% RSLogix 500 project alarm_count.RSS, saved by version 8.30.00.16 %
PROJECT "UNTITLED"    % processor: Bul.1763 MicroLogix 1100 Series B %

PROGRAM FILES
  LAD 2 "MAIN"  4 rungs
  LAD 3 "SUB_AND"  6 rungs
  LAD 4 "PARALLEL"  12 rungs
  LAD 5 "XIC_BRUTEF"  3 rungs
  LAD 6 "LOOKUPBYTE"  5 rungs
  LAD 7 "SUBANDUNRL"  129 rungs
  LAD 254 "WRITE_BITS"  5 rungs
  LAD 255 "BITSPRBYTE"  5 rungs

DATA FILES
  O0 OUTPUT  4 elements
  I1 INPUT  6 elements
  S2 STATUS  66 elements
  B3 BINARY  3 elements
  T4 TIMER  11 elements
  C5 COUNTER  1 elements
  R6 CONTROL  1 elements
  N7 INTEGER  10 elements
  F8 FLOAT  4 elements
  L9 LONG_DATA  12 elements
  N10 BITSPRBYTE  256 elements
  L11 LONG_MASKS  12 elements
  L100 CONTRLTIME  256 elements
  L101 SUBANDTIME  256 elements
  L102 PARLLLTIME  256 elements
  L103 XIC_TIME  256 elements
  L104 LOOKUPTIME  256 elements
  L105 SUBANDUNRL  256 elements

LADDER 2 "MAIN"
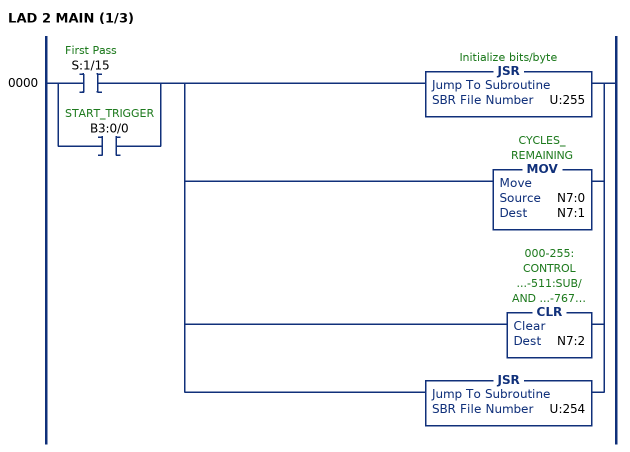
% Rung: 0 %
SOR BST XIC S:1/15 NXB XIC B3:0/0 BND BST JSR U:255 NXB MOV N7:0 N7:1 NXB CLR N7:2 NXB JSR U:254 BND EOR
%   S:1/15  "First Pass" %
%   B3:0/0  START_TRIGGER %
%   U:255  "Initialize bits/byte" %
%   N7:0  TEST_CYCLES %
%   N7:1  CYCLES_REMAINING %
%   N7:2  WHICH  "000-255:CONTROL ...-511:SUB/AND ...-767:PARALLEL ...-1023:XIC ...-1279:LOOKUP_BYTE" %

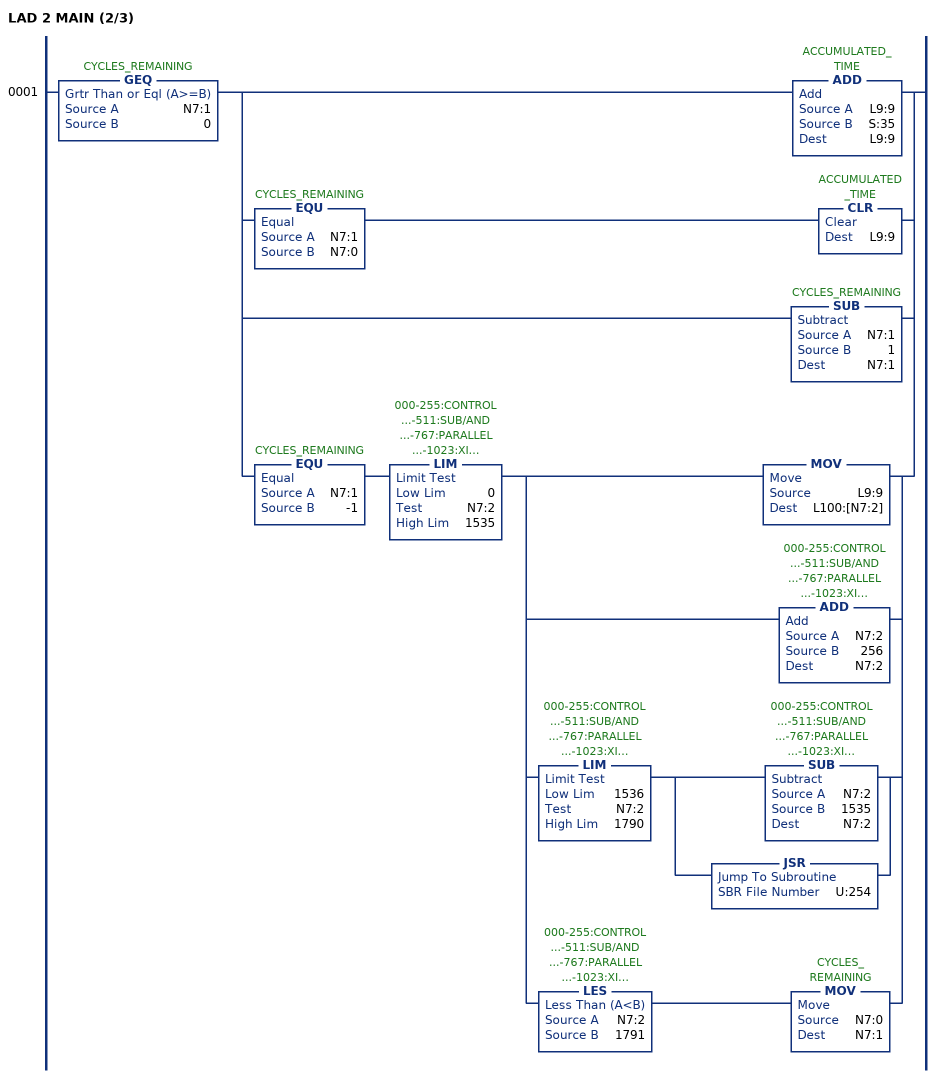
% Rung: 1 %
SOR GEQ N7:1 0 BST ADD L9:9 S:35 L9:9 NXB EQU N7:1 N7:0 CLR L9:9 NXB SUB N7:1 1 N7:1 NXB EQU N7:1 -1 LIM 0 N7:2 1535 BST MOV L9:9 L100:[N7:2] NXB ADD N7:2 256 N7:2 NXB LIM 1536 N7:2 1790 BST SUB N7:2 1535 N7:2 NXB JSR U:254 BND NXB LES N7:2 1791 MOV N7:0 N7:1 BND BND EOR
%   N7:1  CYCLES_REMAINING %
%   L9:9  ACCUMULATED_TIME %
%   S:35  "Last 1 ms Scan Time" %
%   N7:0  TEST_CYCLES %
%   N7:2  WHICH  "000-255:CONTROL ...-511:SUB/AND ...-767:PARALLEL ...-1023:XIC ...-1279:LOOKUP_BYTE" %

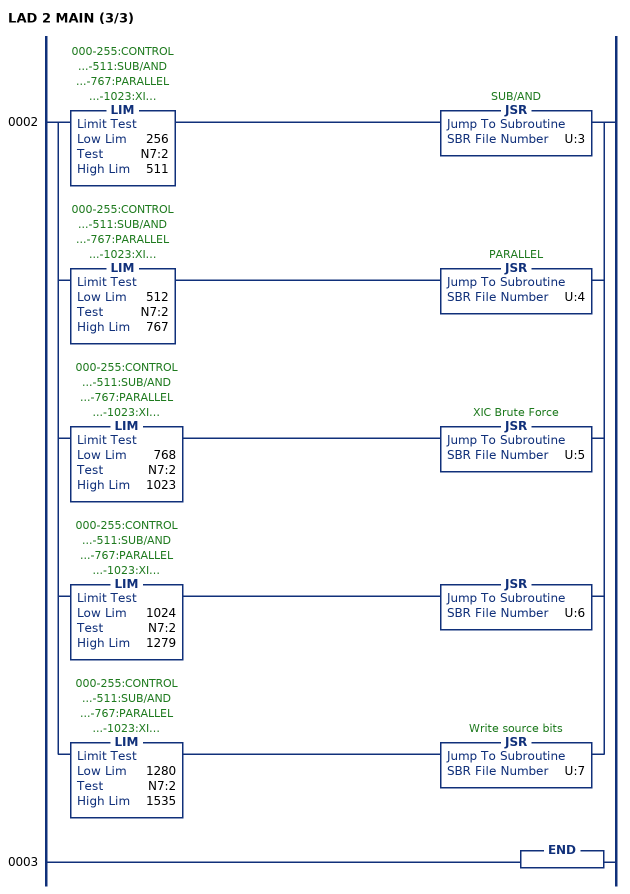
% Rung: 2 %
SOR BST LIM 256 N7:2 511 JSR U:3 NXB LIM 512 N7:2 767 JSR U:4 NXB LIM 768 N7:2 1023 JSR U:5 NXB LIM 1024 N7:2 1279 JSR U:6 NXB LIM 1280 N7:2 1535 JSR U:7 BND EOR
%   N7:2  WHICH  "000-255:CONTROL ...-511:SUB/AND ...-767:PARALLEL ...-1023:XIC ...-1279:LOOKUP_BYTE" %
%   U:3  "SUB/AND" %
%   U:4  "PARALLEL" %
%   U:5  "XIC Brute Force" %
%   U:7  "Write source bits" %
% Rung: 3 %
SOR END EOR

LADDER 3 "SUB_AND"
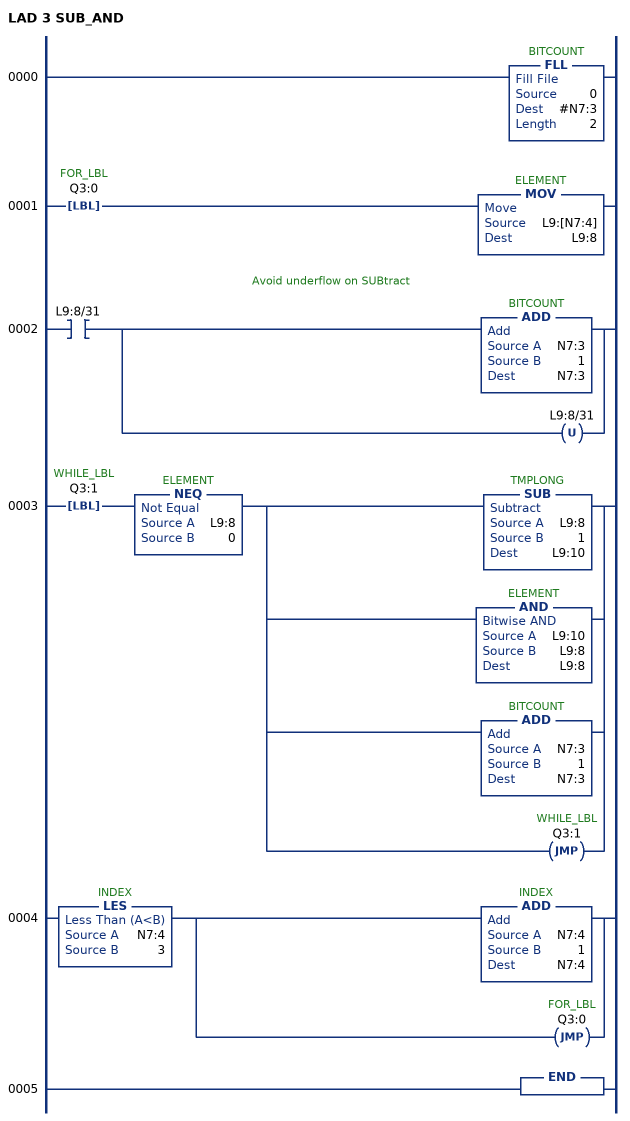
% Rung: 0 %
SOR FLL 0 #N7:3 2 EOR
%   N7:3  BITCOUNT %
% Rung: 1 %
SOR LBL Q3:0 MOV L9:[N7:4] L9:8 EOR
%   Q3:0  FOR_LBL %
%   N7:4  INDEX %
%   L9:8  ELEMENT %
% Rung: 2 %
% Avoid underflow on SUBtract %
SOR XIC L9:8/31 BST ADD N7:3 1 N7:3 NXB OTU L9:8/31 BND EOR
%   N7:3  BITCOUNT %
% Rung: 3 %
SOR LBL Q3:1 NEQ L9:8 0 BST SUB L9:8 1 L9:10 NXB AND L9:10 L9:8 L9:8 NXB ADD N7:3 1 N7:3 NXB JMP Q3:1 BND EOR
%   Q3:1  WHILE_LBL %
%   L9:8  ELEMENT %
%   L9:10  TMPLONG %
%   N7:3  BITCOUNT %
% Rung: 4 %
SOR LES N7:4 3 BST ADD N7:4 1 N7:4 NXB JMP Q3:0 BND EOR
%   N7:4  INDEX %
%   Q3:0  FOR_LBL %
% Rung: 5 %
SOR END EOR

LADDER 4 "PARALLEL"
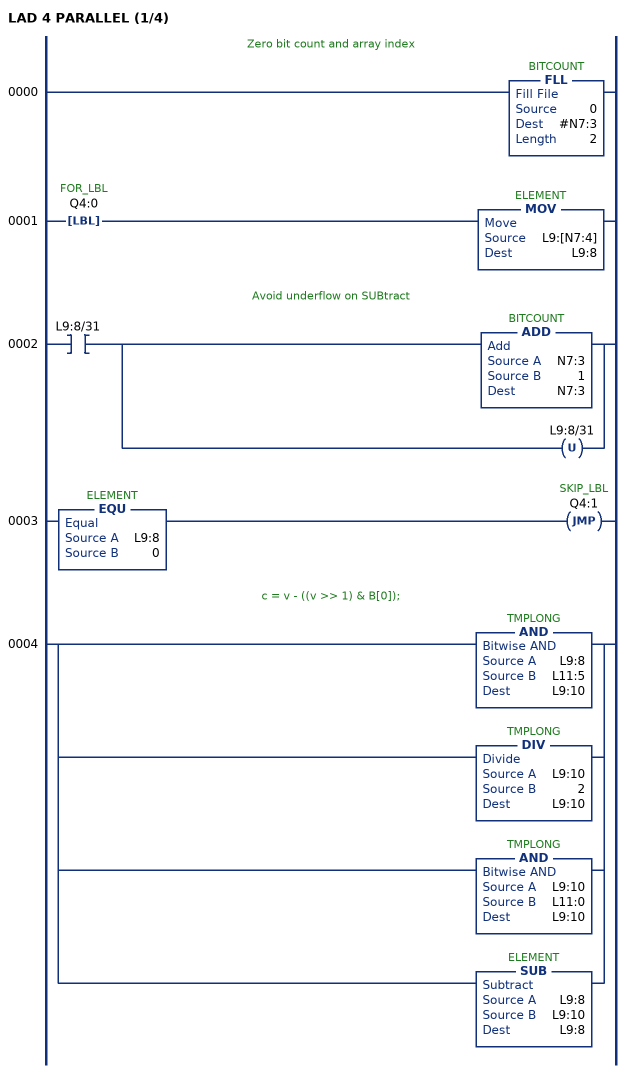
% Rung: 0 %
% Zero bit count and array index %
SOR FLL 0 #N7:3 2 EOR
%   N7:3  BITCOUNT %
% Rung: 1 %
SOR LBL Q4:0 MOV L9:[N7:4] L9:8 EOR
%   Q4:0  "FOR_LBL" %
%   N7:4  INDEX %
%   L9:8  ELEMENT %
% Rung: 2 %
% Avoid underflow on SUBtract %
SOR XIC L9:8/31 BST ADD N7:3 1 N7:3 NXB OTU L9:8/31 BND EOR
%   N7:3  BITCOUNT %
% Rung: 3 %
SOR EQU L9:8 0 JMP Q4:1 EOR
%   L9:8  ELEMENT %
%   Q4:1  "SKIP_LBL" %
% Rung: 4 %
% c = v - ((v >> 1) & B[0]); %
SOR BST AND L9:8 L11:5 L9:10 NXB DIV L9:10 2 L9:10 NXB AND L9:10 L11:0 L9:10 NXB SUB L9:8 L9:10 L9:8 BND EOR
%   L9:8  ELEMENT %
%   L11:5  0XFFFFFFFE_S0 %
%   L9:10  TMPLONG %
%   L11:0  0X55555555_B0 %

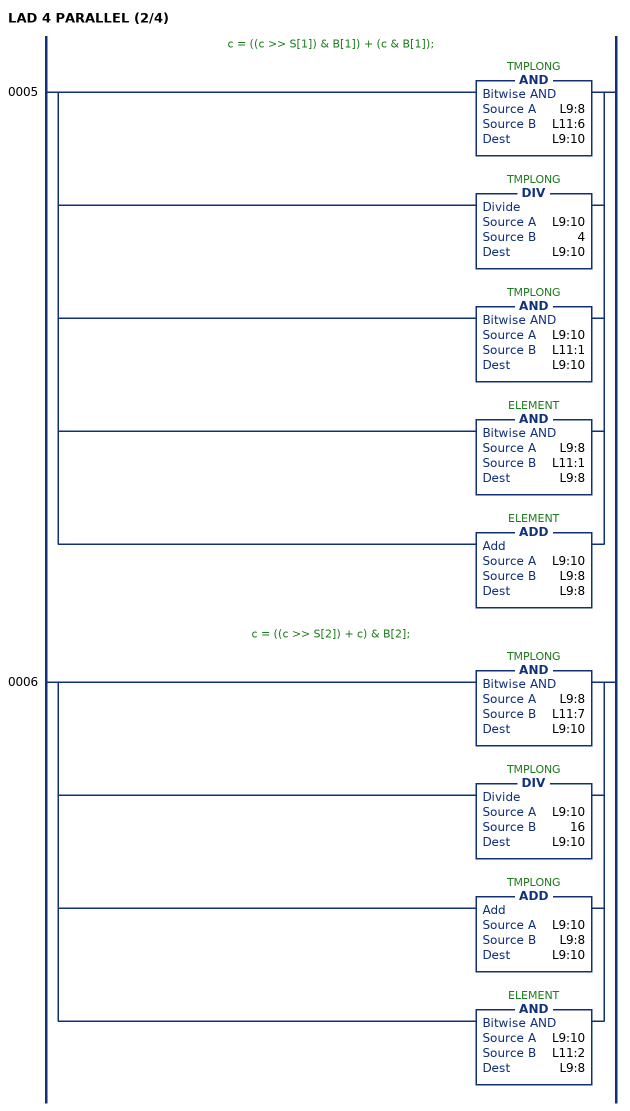
% Rung: 5 %
% c = ((c >> S[1]) & B[1]) + (c & B[1]); %
SOR BST AND L9:8 L11:6 L9:10 NXB DIV L9:10 4 L9:10 NXB AND L9:10 L11:1 L9:10 NXB AND L9:8 L11:1 L9:8 NXB ADD L9:10 L9:8 L9:8 BND EOR
%   L9:8  ELEMENT %
%   L11:6  0XFFFFFFFC_S1 %
%   L9:10  TMPLONG %
%   L11:1  0X33333333_B1 %
% Rung: 6 %
% c = ((c >> S[2]) + c) & B[2]; %
SOR BST AND L9:8 L11:7 L9:10 NXB DIV L9:10 16 L9:10 NXB ADD L9:10 L9:8 L9:10 NXB AND L9:10 L11:2 L9:8 BND EOR
%   L9:8  ELEMENT %
%   L11:7  0XFFFFFFF0_S2 %
%   L9:10  TMPLONG %
%   L11:2  0X0F0F0F0F_B2 %

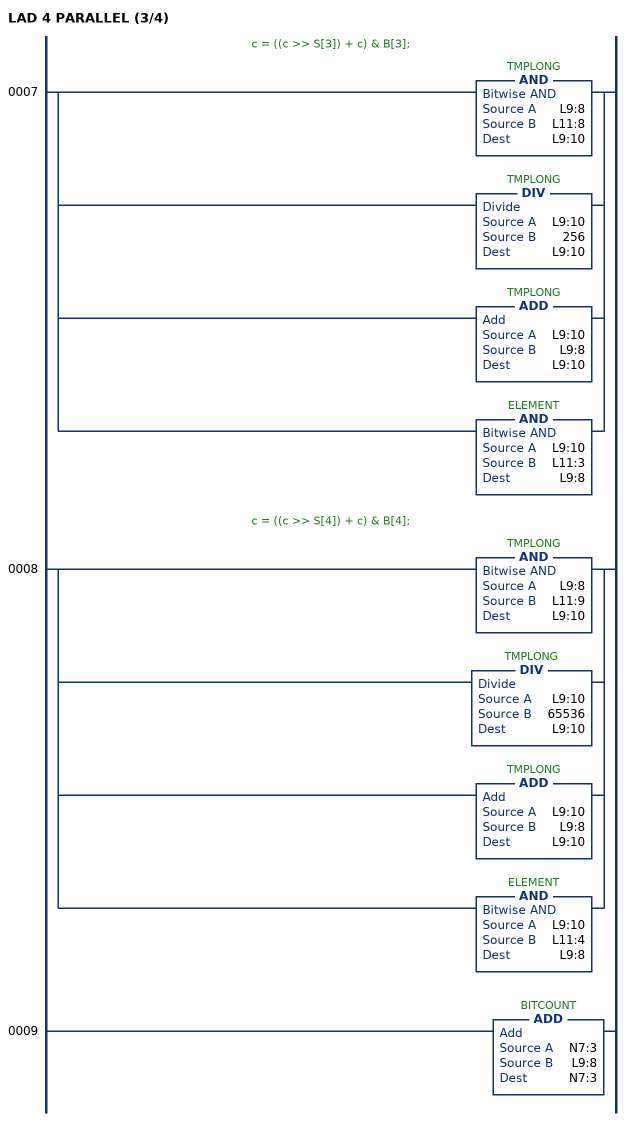
% Rung: 7 %
% c = ((c >> S[3]) + c) & B[3]; %
SOR BST AND L9:8 L11:8 L9:10 NXB DIV L9:10 256 L9:10 NXB ADD L9:10 L9:8 L9:10 NXB AND L9:10 L11:3 L9:8 BND EOR
%   L9:8  ELEMENT %
%   L11:8  0XFFFFFF00_S3 %
%   L9:10  TMPLONG %
%   L11:3  0X00FF00FF_B3 %
% Rung: 8 %
% c = ((c >> S[4]) + c) & B[4]; %
SOR BST AND L9:8 L11:9 L9:10 NXB DIV L9:10 65536 L9:10 NXB ADD L9:10 L9:8 L9:10 NXB AND L9:10 L11:4 L9:8 BND EOR
%   L9:8  ELEMENT %
%   L11:9  0XFFFF0000_S4 %
%   L9:10  TMPLONG %
%   L11:4  0X0000FFFF_B4 %
% Rung: 9 %
SOR ADD N7:3 L9:8 N7:3 EOR
%   N7:3  BITCOUNT %
%   L9:8  ELEMENT %

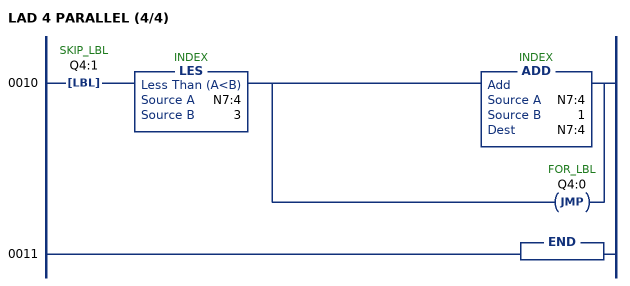
% Rung: 10 %
SOR LBL Q4:1 LES N7:4 3 BST ADD N7:4 1 N7:4 NXB JMP Q4:0 BND EOR
%   Q4:1  "SKIP_LBL" %
%   N7:4  INDEX %
%   Q4:0  "FOR_LBL" %
% Rung: 11 %
SOR END EOR

LADDER 5 "XIC_BRUTEF"
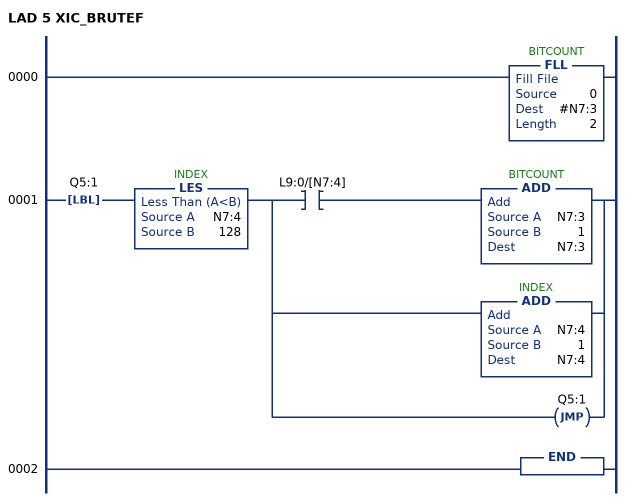
% Rung: 0 %
SOR FLL 0 #N7:3 2 EOR
%   N7:3  BITCOUNT %
% Rung: 1 %
SOR LBL Q5:1 LES N7:4 128 BST XIC L9:0/[N7:4] ADD N7:3 1 N7:3 NXB ADD N7:4 1 N7:4 NXB JMP Q5:1 BND EOR
%   N7:4  INDEX %
%   L9:0  128_SOURCE_BITS %
%   N7:3  BITCOUNT %
% Rung: 2 %
SOR END EOR

LADDER 6 "LOOKUPBYTE"
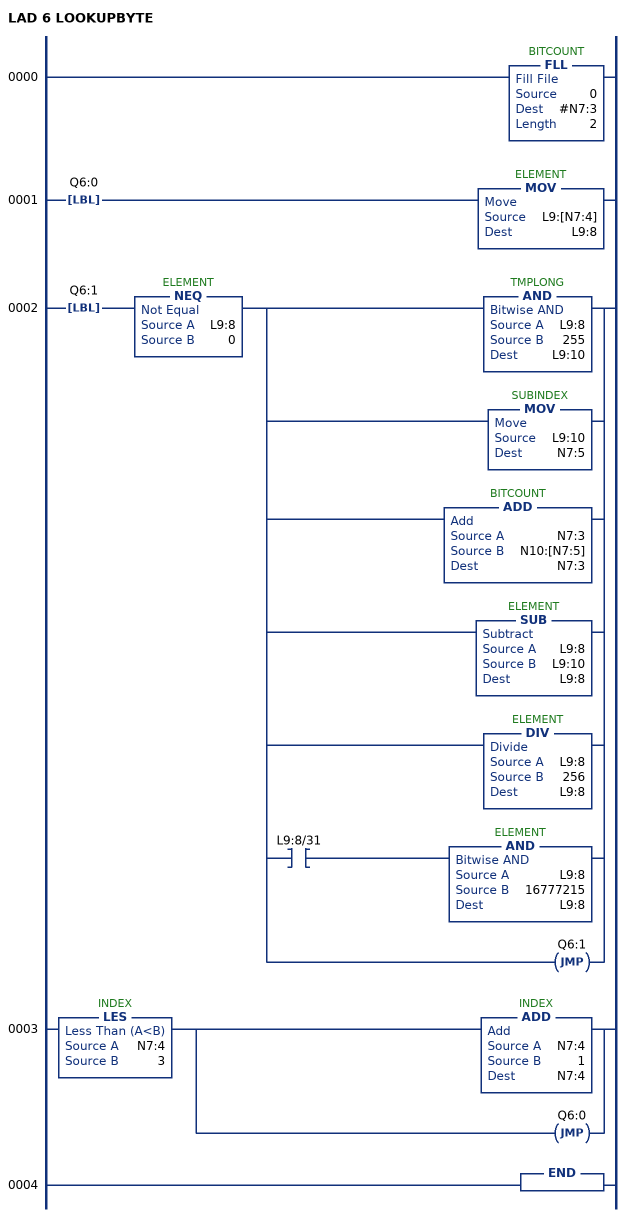
% Rung: 0 %
SOR FLL 0 #N7:3 2 EOR
%   N7:3  BITCOUNT %
% Rung: 1 %
SOR LBL Q6:0 MOV L9:[N7:4] L9:8 EOR
%   N7:4  INDEX %
%   L9:8  ELEMENT %
% Rung: 2 %
SOR LBL Q6:1 NEQ L9:8 0 BST AND L9:8 255 L9:10 NXB MOV L9:10 N7:5 NXB ADD N7:3 N10:[N7:5] N7:3 NXB SUB L9:8 L9:10 L9:8 NXB DIV L9:8 256 L9:8 NXB XIC L9:8/31 AND L9:8 16777215 L9:8 NXB JMP Q6:1 BND EOR
%   L9:8  ELEMENT %
%   L9:10  TMPLONG %
%   N7:5  SUBINDEX %
%   N7:3  BITCOUNT %
% Rung: 3 %
SOR LES N7:4 3 BST ADD N7:4 1 N7:4 NXB JMP Q6:0 BND EOR
%   N7:4  INDEX %
% Rung: 4 %
SOR END EOR

LADDER 7 "SUBANDUNRL"
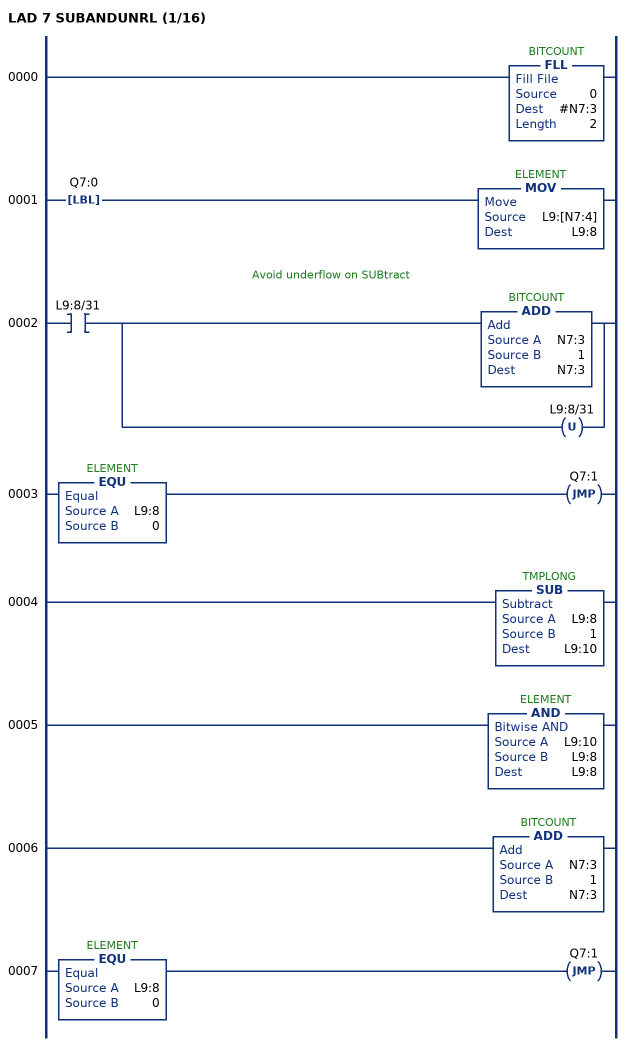
% Rung: 0 %
SOR FLL 0 #N7:3 2 EOR
%   N7:3  BITCOUNT %
% Rung: 1 %
SOR LBL Q7:0 MOV L9:[N7:4] L9:8 EOR
%   N7:4  INDEX %
%   L9:8  ELEMENT %
% Rung: 2 %
% Avoid underflow on SUBtract %
SOR XIC L9:8/31 BST ADD N7:3 1 N7:3 NXB OTU L9:8/31 BND EOR
%   N7:3  BITCOUNT %
% Rung: 3 %
SOR EQU L9:8 0 JMP Q7:1 EOR
%   L9:8  ELEMENT %
% Rung: 4 %
SOR SUB L9:8 1 L9:10 EOR
%   L9:8  ELEMENT %
%   L9:10  TMPLONG %
% Rung: 5 %
SOR AND L9:10 L9:8 L9:8 EOR
%   L9:10  TMPLONG %
%   L9:8  ELEMENT %
% Rung: 6 %
SOR ADD N7:3 1 N7:3 EOR
%   N7:3  BITCOUNT %
% Rung: 7 %
SOR EQU L9:8 0 JMP Q7:1 EOR
%   L9:8  ELEMENT %

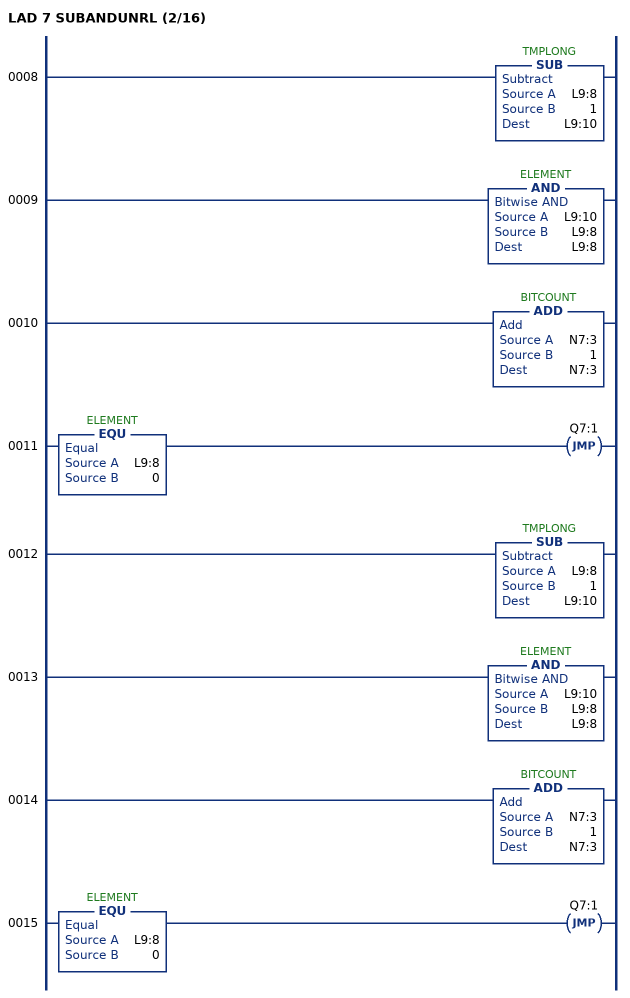
% Rung: 8 %
SOR SUB L9:8 1 L9:10 EOR
%   L9:8  ELEMENT %
%   L9:10  TMPLONG %
% Rung: 9 %
SOR AND L9:10 L9:8 L9:8 EOR
%   L9:10  TMPLONG %
%   L9:8  ELEMENT %
% Rung: 10 %
SOR ADD N7:3 1 N7:3 EOR
%   N7:3  BITCOUNT %
% Rung: 11 %
SOR EQU L9:8 0 JMP Q7:1 EOR
%   L9:8  ELEMENT %
% Rung: 12 %
SOR SUB L9:8 1 L9:10 EOR
%   L9:8  ELEMENT %
%   L9:10  TMPLONG %
% Rung: 13 %
SOR AND L9:10 L9:8 L9:8 EOR
%   L9:10  TMPLONG %
%   L9:8  ELEMENT %
% Rung: 14 %
SOR ADD N7:3 1 N7:3 EOR
%   N7:3  BITCOUNT %
% Rung: 15 %
SOR EQU L9:8 0 JMP Q7:1 EOR
%   L9:8  ELEMENT %

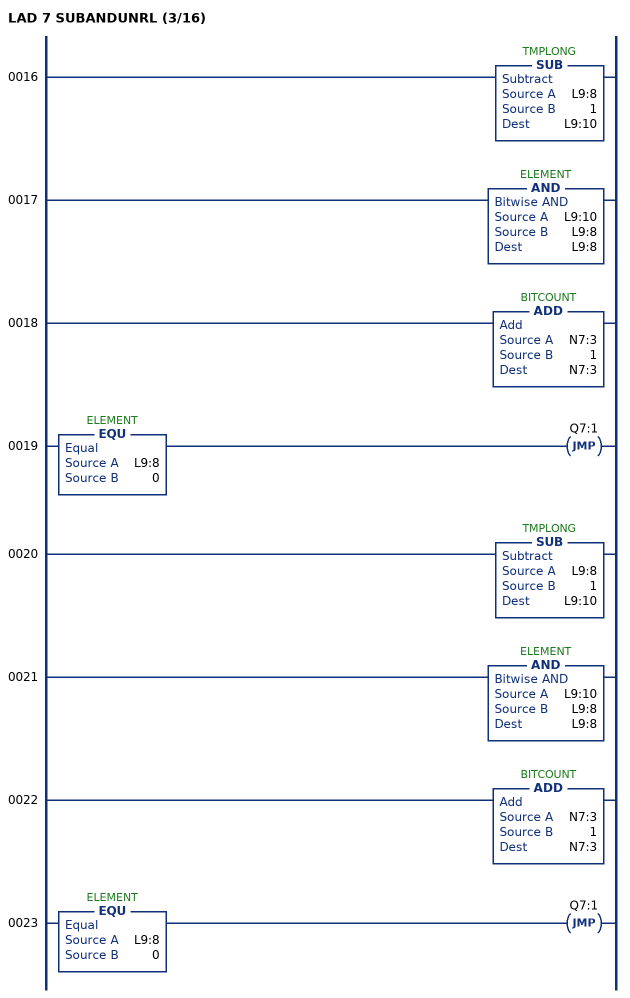
% Rung: 16 %
SOR SUB L9:8 1 L9:10 EOR
%   L9:8  ELEMENT %
%   L9:10  TMPLONG %
% Rung: 17 %
SOR AND L9:10 L9:8 L9:8 EOR
%   L9:10  TMPLONG %
%   L9:8  ELEMENT %
% Rung: 18 %
SOR ADD N7:3 1 N7:3 EOR
%   N7:3  BITCOUNT %
% Rung: 19 %
SOR EQU L9:8 0 JMP Q7:1 EOR
%   L9:8  ELEMENT %
% Rung: 20 %
SOR SUB L9:8 1 L9:10 EOR
%   L9:8  ELEMENT %
%   L9:10  TMPLONG %
% Rung: 21 %
SOR AND L9:10 L9:8 L9:8 EOR
%   L9:10  TMPLONG %
%   L9:8  ELEMENT %
% Rung: 22 %
SOR ADD N7:3 1 N7:3 EOR
%   N7:3  BITCOUNT %
% Rung: 23 %
SOR EQU L9:8 0 JMP Q7:1 EOR
%   L9:8  ELEMENT %

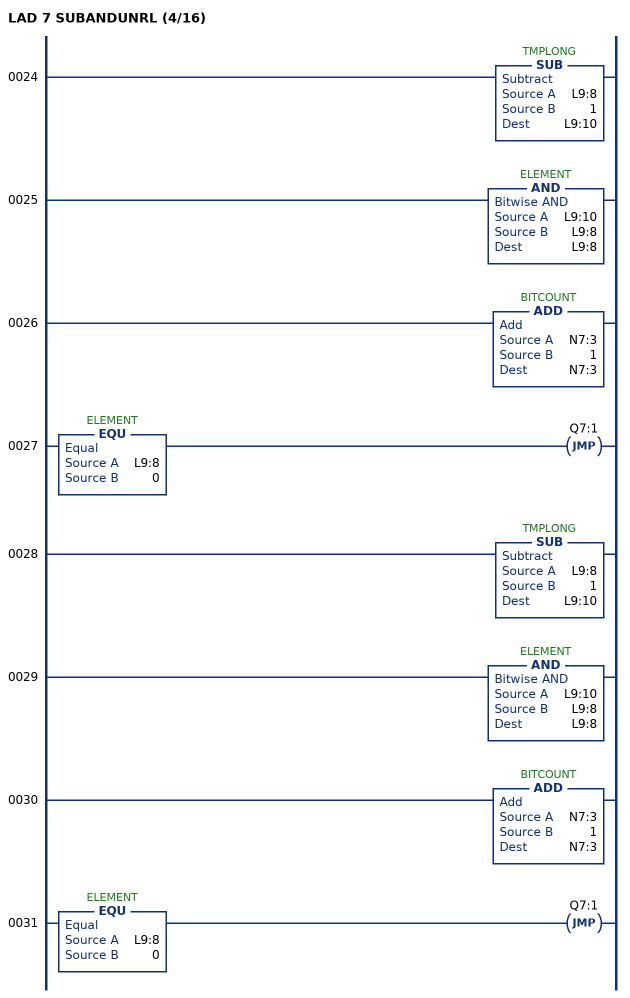
% Rung: 24 %
SOR SUB L9:8 1 L9:10 EOR
%   L9:8  ELEMENT %
%   L9:10  TMPLONG %
% Rung: 25 %
SOR AND L9:10 L9:8 L9:8 EOR
%   L9:10  TMPLONG %
%   L9:8  ELEMENT %
% Rung: 26 %
SOR ADD N7:3 1 N7:3 EOR
%   N7:3  BITCOUNT %
% Rung: 27 %
SOR EQU L9:8 0 JMP Q7:1 EOR
%   L9:8  ELEMENT %
% Rung: 28 %
SOR SUB L9:8 1 L9:10 EOR
%   L9:8  ELEMENT %
%   L9:10  TMPLONG %
% Rung: 29 %
SOR AND L9:10 L9:8 L9:8 EOR
%   L9:10  TMPLONG %
%   L9:8  ELEMENT %
% Rung: 30 %
SOR ADD N7:3 1 N7:3 EOR
%   N7:3  BITCOUNT %
% Rung: 31 %
SOR EQU L9:8 0 JMP Q7:1 EOR
%   L9:8  ELEMENT %

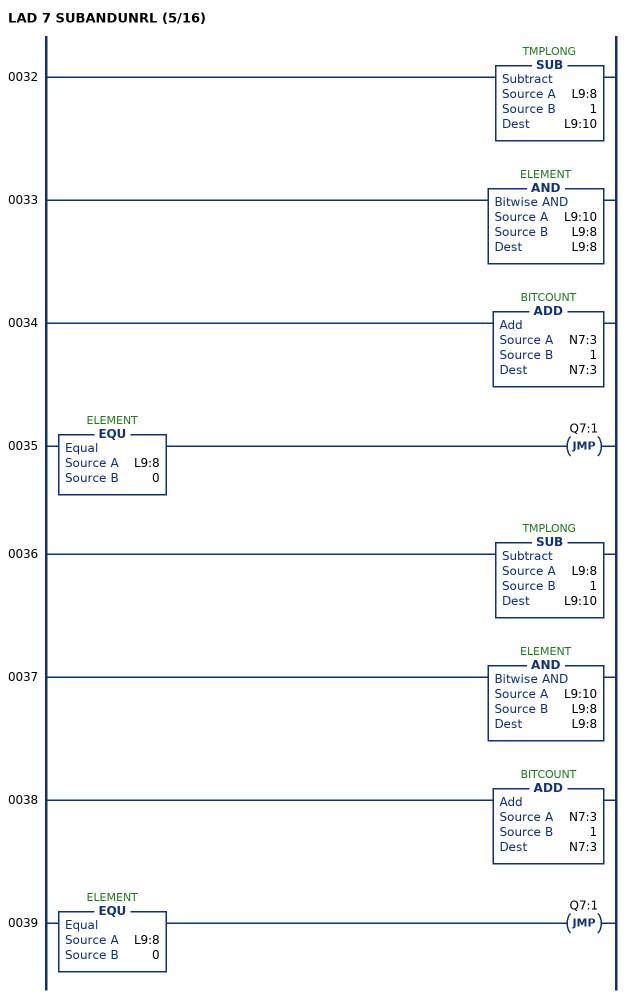
% Rung: 32 %
SOR SUB L9:8 1 L9:10 EOR
%   L9:8  ELEMENT %
%   L9:10  TMPLONG %
% Rung: 33 %
SOR AND L9:10 L9:8 L9:8 EOR
%   L9:10  TMPLONG %
%   L9:8  ELEMENT %
% Rung: 34 %
SOR ADD N7:3 1 N7:3 EOR
%   N7:3  BITCOUNT %
% Rung: 35 %
SOR EQU L9:8 0 JMP Q7:1 EOR
%   L9:8  ELEMENT %
% Rung: 36 %
SOR SUB L9:8 1 L9:10 EOR
%   L9:8  ELEMENT %
%   L9:10  TMPLONG %
% Rung: 37 %
SOR AND L9:10 L9:8 L9:8 EOR
%   L9:10  TMPLONG %
%   L9:8  ELEMENT %
% Rung: 38 %
SOR ADD N7:3 1 N7:3 EOR
%   N7:3  BITCOUNT %
% Rung: 39 %
SOR EQU L9:8 0 JMP Q7:1 EOR
%   L9:8  ELEMENT %

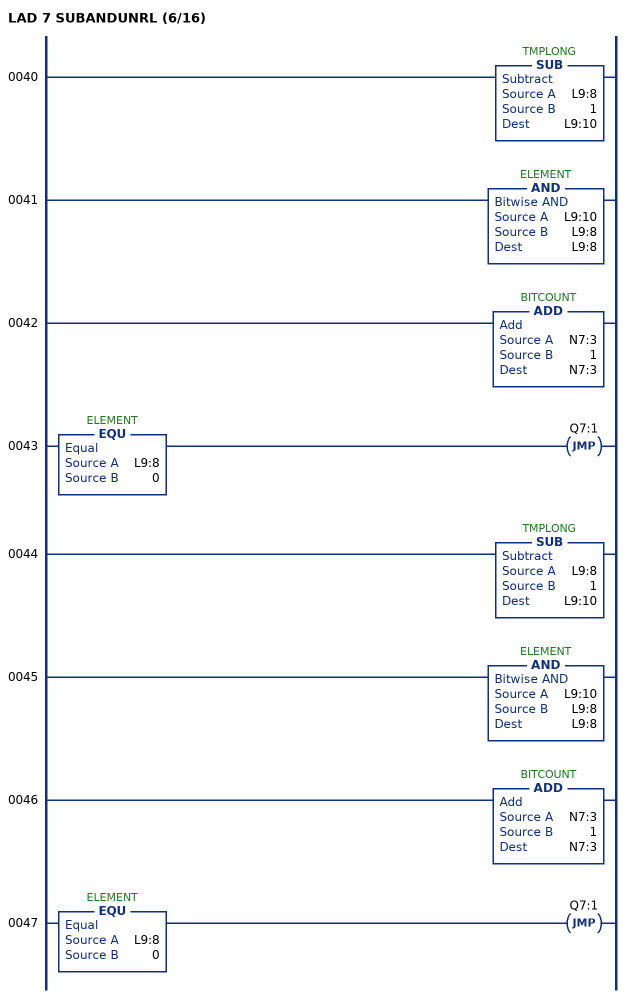
% Rung: 40 %
SOR SUB L9:8 1 L9:10 EOR
%   L9:8  ELEMENT %
%   L9:10  TMPLONG %
% Rung: 41 %
SOR AND L9:10 L9:8 L9:8 EOR
%   L9:10  TMPLONG %
%   L9:8  ELEMENT %
% Rung: 42 %
SOR ADD N7:3 1 N7:3 EOR
%   N7:3  BITCOUNT %
% Rung: 43 %
SOR EQU L9:8 0 JMP Q7:1 EOR
%   L9:8  ELEMENT %
% Rung: 44 %
SOR SUB L9:8 1 L9:10 EOR
%   L9:8  ELEMENT %
%   L9:10  TMPLONG %
% Rung: 45 %
SOR AND L9:10 L9:8 L9:8 EOR
%   L9:10  TMPLONG %
%   L9:8  ELEMENT %
% Rung: 46 %
SOR ADD N7:3 1 N7:3 EOR
%   N7:3  BITCOUNT %
% Rung: 47 %
SOR EQU L9:8 0 JMP Q7:1 EOR
%   L9:8  ELEMENT %

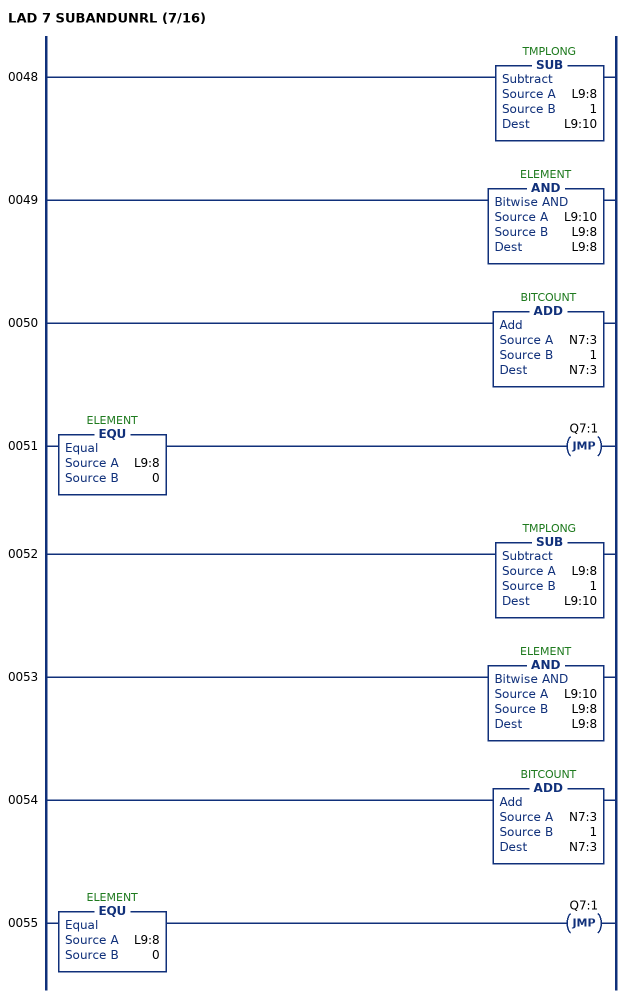
% Rung: 48 %
SOR SUB L9:8 1 L9:10 EOR
%   L9:8  ELEMENT %
%   L9:10  TMPLONG %
% Rung: 49 %
SOR AND L9:10 L9:8 L9:8 EOR
%   L9:10  TMPLONG %
%   L9:8  ELEMENT %
% Rung: 50 %
SOR ADD N7:3 1 N7:3 EOR
%   N7:3  BITCOUNT %
% Rung: 51 %
SOR EQU L9:8 0 JMP Q7:1 EOR
%   L9:8  ELEMENT %
% Rung: 52 %
SOR SUB L9:8 1 L9:10 EOR
%   L9:8  ELEMENT %
%   L9:10  TMPLONG %
% Rung: 53 %
SOR AND L9:10 L9:8 L9:8 EOR
%   L9:10  TMPLONG %
%   L9:8  ELEMENT %
% Rung: 54 %
SOR ADD N7:3 1 N7:3 EOR
%   N7:3  BITCOUNT %
% Rung: 55 %
SOR EQU L9:8 0 JMP Q7:1 EOR
%   L9:8  ELEMENT %

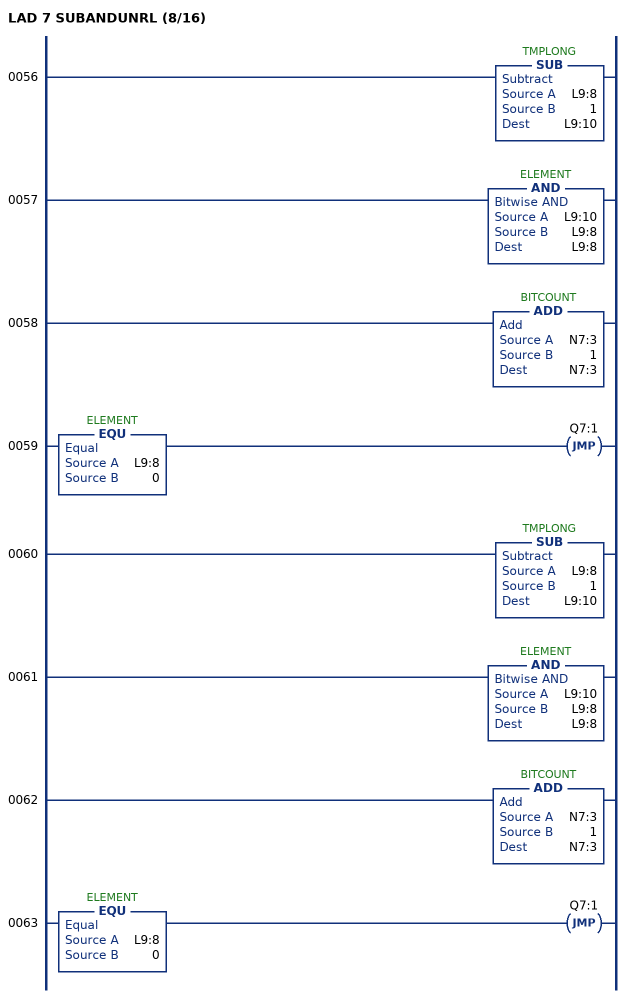
% Rung: 56 %
SOR SUB L9:8 1 L9:10 EOR
%   L9:8  ELEMENT %
%   L9:10  TMPLONG %
% Rung: 57 %
SOR AND L9:10 L9:8 L9:8 EOR
%   L9:10  TMPLONG %
%   L9:8  ELEMENT %
% Rung: 58 %
SOR ADD N7:3 1 N7:3 EOR
%   N7:3  BITCOUNT %
% Rung: 59 %
SOR EQU L9:8 0 JMP Q7:1 EOR
%   L9:8  ELEMENT %
% Rung: 60 %
SOR SUB L9:8 1 L9:10 EOR
%   L9:8  ELEMENT %
%   L9:10  TMPLONG %
% Rung: 61 %
SOR AND L9:10 L9:8 L9:8 EOR
%   L9:10  TMPLONG %
%   L9:8  ELEMENT %
% Rung: 62 %
SOR ADD N7:3 1 N7:3 EOR
%   N7:3  BITCOUNT %
% Rung: 63 %
SOR EQU L9:8 0 JMP Q7:1 EOR
%   L9:8  ELEMENT %

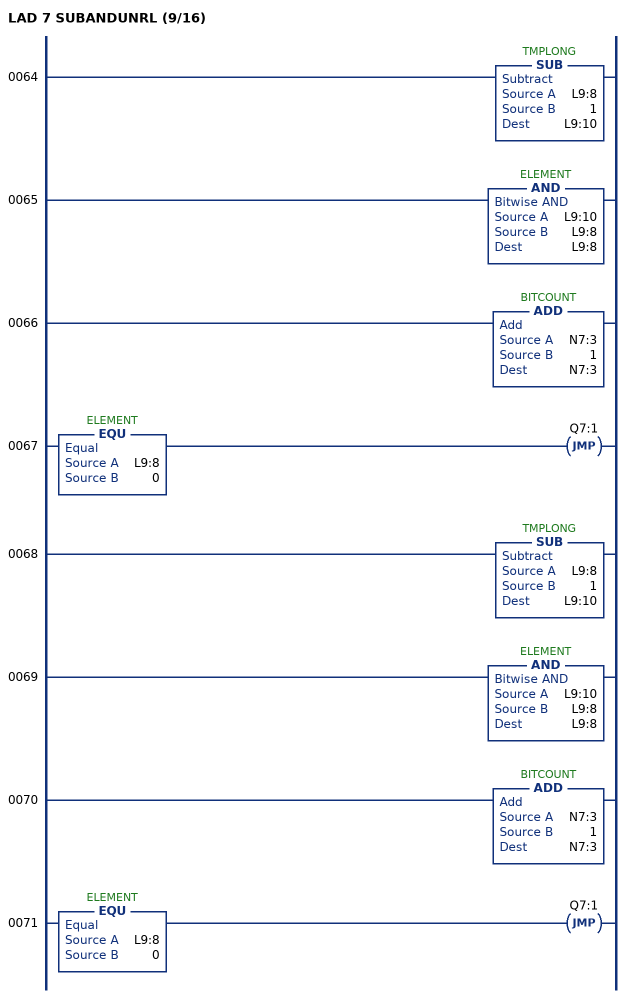
% Rung: 64 %
SOR SUB L9:8 1 L9:10 EOR
%   L9:8  ELEMENT %
%   L9:10  TMPLONG %
% Rung: 65 %
SOR AND L9:10 L9:8 L9:8 EOR
%   L9:10  TMPLONG %
%   L9:8  ELEMENT %
% Rung: 66 %
SOR ADD N7:3 1 N7:3 EOR
%   N7:3  BITCOUNT %
% Rung: 67 %
SOR EQU L9:8 0 JMP Q7:1 EOR
%   L9:8  ELEMENT %
% Rung: 68 %
SOR SUB L9:8 1 L9:10 EOR
%   L9:8  ELEMENT %
%   L9:10  TMPLONG %
% Rung: 69 %
SOR AND L9:10 L9:8 L9:8 EOR
%   L9:10  TMPLONG %
%   L9:8  ELEMENT %
% Rung: 70 %
SOR ADD N7:3 1 N7:3 EOR
%   N7:3  BITCOUNT %
% Rung: 71 %
SOR EQU L9:8 0 JMP Q7:1 EOR
%   L9:8  ELEMENT %

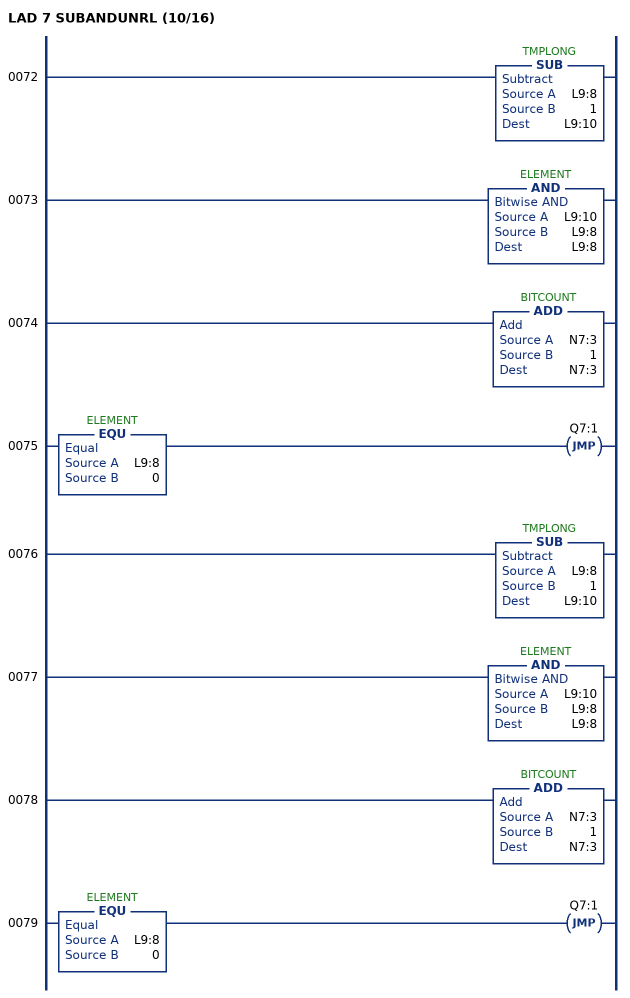
% Rung: 72 %
SOR SUB L9:8 1 L9:10 EOR
%   L9:8  ELEMENT %
%   L9:10  TMPLONG %
% Rung: 73 %
SOR AND L9:10 L9:8 L9:8 EOR
%   L9:10  TMPLONG %
%   L9:8  ELEMENT %
% Rung: 74 %
SOR ADD N7:3 1 N7:3 EOR
%   N7:3  BITCOUNT %
% Rung: 75 %
SOR EQU L9:8 0 JMP Q7:1 EOR
%   L9:8  ELEMENT %
% Rung: 76 %
SOR SUB L9:8 1 L9:10 EOR
%   L9:8  ELEMENT %
%   L9:10  TMPLONG %
% Rung: 77 %
SOR AND L9:10 L9:8 L9:8 EOR
%   L9:10  TMPLONG %
%   L9:8  ELEMENT %
% Rung: 78 %
SOR ADD N7:3 1 N7:3 EOR
%   N7:3  BITCOUNT %
% Rung: 79 %
SOR EQU L9:8 0 JMP Q7:1 EOR
%   L9:8  ELEMENT %

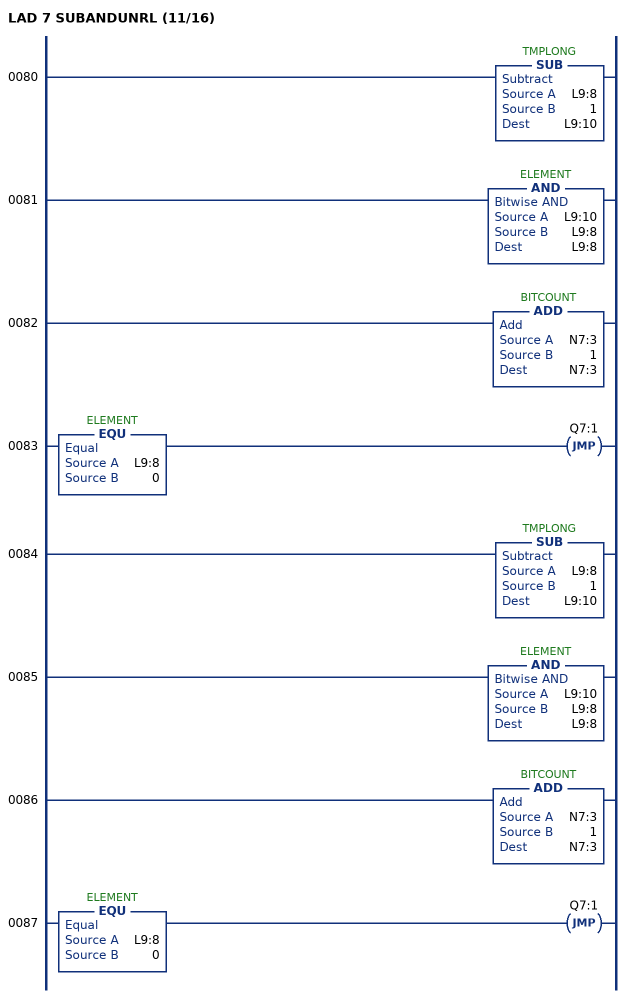
% Rung: 80 %
SOR SUB L9:8 1 L9:10 EOR
%   L9:8  ELEMENT %
%   L9:10  TMPLONG %
% Rung: 81 %
SOR AND L9:10 L9:8 L9:8 EOR
%   L9:10  TMPLONG %
%   L9:8  ELEMENT %
% Rung: 82 %
SOR ADD N7:3 1 N7:3 EOR
%   N7:3  BITCOUNT %
% Rung: 83 %
SOR EQU L9:8 0 JMP Q7:1 EOR
%   L9:8  ELEMENT %
% Rung: 84 %
SOR SUB L9:8 1 L9:10 EOR
%   L9:8  ELEMENT %
%   L9:10  TMPLONG %
% Rung: 85 %
SOR AND L9:10 L9:8 L9:8 EOR
%   L9:10  TMPLONG %
%   L9:8  ELEMENT %
% Rung: 86 %
SOR ADD N7:3 1 N7:3 EOR
%   N7:3  BITCOUNT %
% Rung: 87 %
SOR EQU L9:8 0 JMP Q7:1 EOR
%   L9:8  ELEMENT %

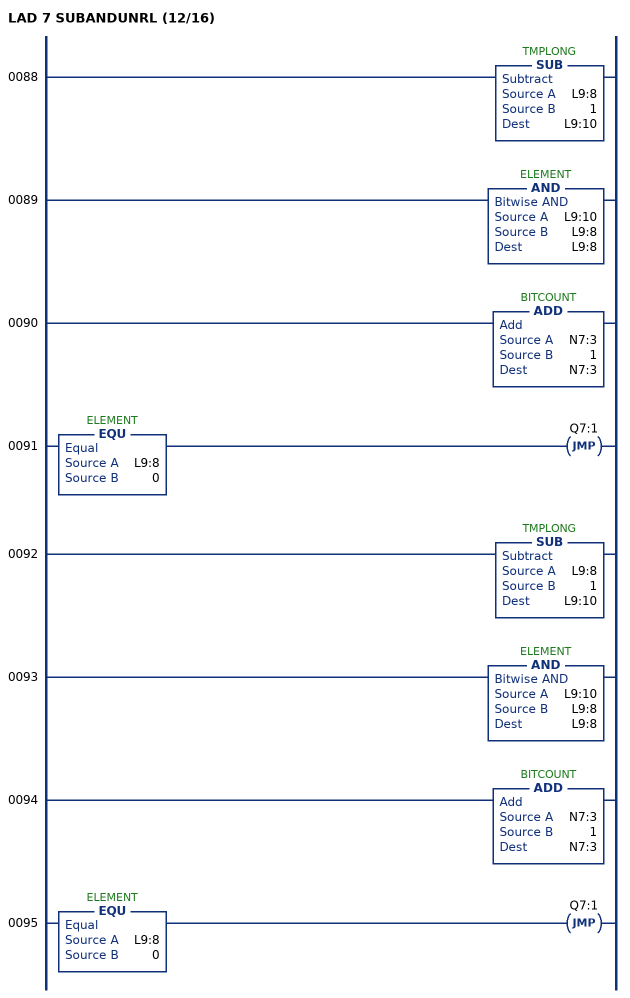
% Rung: 88 %
SOR SUB L9:8 1 L9:10 EOR
%   L9:8  ELEMENT %
%   L9:10  TMPLONG %
% Rung: 89 %
SOR AND L9:10 L9:8 L9:8 EOR
%   L9:10  TMPLONG %
%   L9:8  ELEMENT %
% Rung: 90 %
SOR ADD N7:3 1 N7:3 EOR
%   N7:3  BITCOUNT %
% Rung: 91 %
SOR EQU L9:8 0 JMP Q7:1 EOR
%   L9:8  ELEMENT %
% Rung: 92 %
SOR SUB L9:8 1 L9:10 EOR
%   L9:8  ELEMENT %
%   L9:10  TMPLONG %
% Rung: 93 %
SOR AND L9:10 L9:8 L9:8 EOR
%   L9:10  TMPLONG %
%   L9:8  ELEMENT %
% Rung: 94 %
SOR ADD N7:3 1 N7:3 EOR
%   N7:3  BITCOUNT %
% Rung: 95 %
SOR EQU L9:8 0 JMP Q7:1 EOR
%   L9:8  ELEMENT %

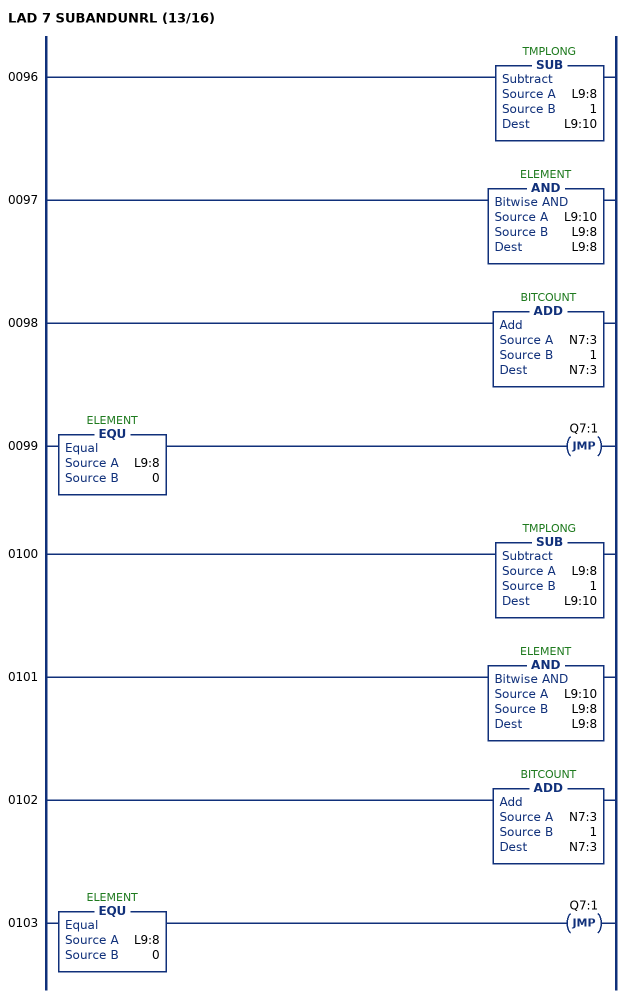
% Rung: 96 %
SOR SUB L9:8 1 L9:10 EOR
%   L9:8  ELEMENT %
%   L9:10  TMPLONG %
% Rung: 97 %
SOR AND L9:10 L9:8 L9:8 EOR
%   L9:10  TMPLONG %
%   L9:8  ELEMENT %
% Rung: 98 %
SOR ADD N7:3 1 N7:3 EOR
%   N7:3  BITCOUNT %
% Rung: 99 %
SOR EQU L9:8 0 JMP Q7:1 EOR
%   L9:8  ELEMENT %
% Rung: 100 %
SOR SUB L9:8 1 L9:10 EOR
%   L9:8  ELEMENT %
%   L9:10  TMPLONG %
% Rung: 101 %
SOR AND L9:10 L9:8 L9:8 EOR
%   L9:10  TMPLONG %
%   L9:8  ELEMENT %
% Rung: 102 %
SOR ADD N7:3 1 N7:3 EOR
%   N7:3  BITCOUNT %
% Rung: 103 %
SOR EQU L9:8 0 JMP Q7:1 EOR
%   L9:8  ELEMENT %

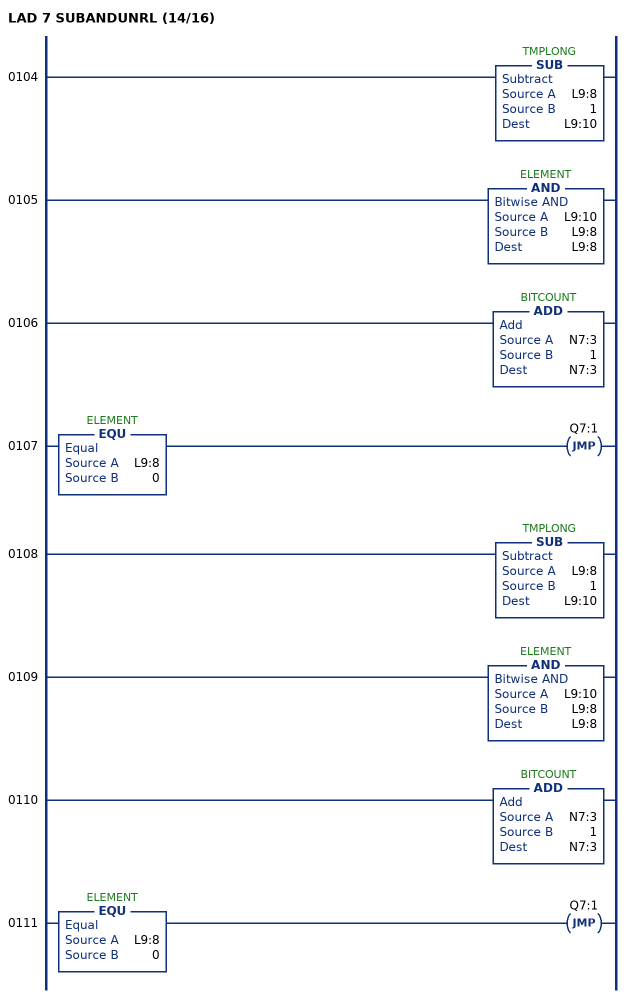
% Rung: 104 %
SOR SUB L9:8 1 L9:10 EOR
%   L9:8  ELEMENT %
%   L9:10  TMPLONG %
% Rung: 105 %
SOR AND L9:10 L9:8 L9:8 EOR
%   L9:10  TMPLONG %
%   L9:8  ELEMENT %
% Rung: 106 %
SOR ADD N7:3 1 N7:3 EOR
%   N7:3  BITCOUNT %
% Rung: 107 %
SOR EQU L9:8 0 JMP Q7:1 EOR
%   L9:8  ELEMENT %
% Rung: 108 %
SOR SUB L9:8 1 L9:10 EOR
%   L9:8  ELEMENT %
%   L9:10  TMPLONG %
% Rung: 109 %
SOR AND L9:10 L9:8 L9:8 EOR
%   L9:10  TMPLONG %
%   L9:8  ELEMENT %
% Rung: 110 %
SOR ADD N7:3 1 N7:3 EOR
%   N7:3  BITCOUNT %
% Rung: 111 %
SOR EQU L9:8 0 JMP Q7:1 EOR
%   L9:8  ELEMENT %

